PROGRAM MAIN
VAR
END_VAR

END_PROGRAM

(* stored: Version 1.1.0.1, ProductVersion 3.1.4024.12
   POU MAIN: Id {6b025910-8a5d-09ab-03d5-eb72258e4660}, SpecialFunc None *)
